{attribute 'enable_dynamic_creation'}
FUNCTION_BLOCK FB_DBTransactionHandler
VAR_INPUT
	ProjectDBDefs : IProjectDBDefs; //Instance of the custom database FB for this database
END_VAR
VAR_OUTPUT
END_VAR
VAR
	//Property backing variables
	_JRSQLNetId : T_AmsNetID;
	_JRSQLPort : T_AmsPort;
	_DBServer : POINTER TO fb_dbserver;
	_Busy : BOOL;
	_Done : BOOL;
	_Error : BOOL;
	_ErrorId : UINT;	
	_ErrorText : STRING;
	
	//'Framework'
	bFirstScan: BOOL := TRUE;
	tmrState:  TON;

	nState:	UDINT	:= 0;
	nNextState:	UDINT	:= 0;
	bFirstEntry: BOOL;	
	
	//Locals
	Triggered : BOOL := FALSE;
	DataReturn : BOOL := FALSE;
	
	spName :STRING;
	spData: pvoid;
	spDataSize:UDINT;
	
	spDefinition : DBSPDefinition;
	spCallResult : DBSPCallResult;
	
	TransmitBuffer : POINTER TO BYTE;
	TransmitSize : UINT;
	ReceiveBuffer : POINTER TO BYTE;
	ReceiveSize : UINT;
	
	LastProcessTime : TIME;
		
	fbADSReadWrite: ADSRDWRTEX;

END_VAR
VAR CONSTANT
	cJRSQLTimeout : TIME := T#10S;
	cJRSQLCommandExecute : UDINT := 16#1000;
END_VAR

IF bFirstScan THEN
	nNextState:=0;
	nState:=9999;
	
	fbADSReadWrite(NETID:=_JRSQLNetId,PORT:=_JRSQLPort,WRTRD:=FALSE,TMOUT:=cJRSQLTimeout);
	bFirstScan := FALSE;
END_IF

//state machine	
IF nState <> nNextState THEN
	bFirstEntry := TRUE;
	nState := nNextState;
ELSE
	bFirstEntry := FALSE;
END_IF

tmrState(IN:=(NOT bFirstEntry), PT:=T#20S);

CASE nState OF
0:
	IF bFirstEntry THEN
		_Error:=FALSE;
		_ErrorId := 16#0;
		_ErrorText := '';
		_Done:=FALSE;
	END_IF

	IF Triggered THEN
		IF _DBServer^.Connected THEN
			nNextState := 40;
		ELSE
			nNextState := 10;
		END_IF
	END_IF
	
10://wait for connection
	IF (_DBServer^.Connected) THEN
		nNextState := 0;
	ELSIF tmrState.ET > cJRSQLTimeout THEN
		_ErrorText:='JRSQL connection timeout';		
		_ErrorId := 16#1;
		_Error:=TRUE;
		nNextState	:= 999;
 	END_IF

//States combined to get rid of scan delays	
40: //Call JRSQL
	IF bFirstEntry THEN
		IF(ProjectDBDefs.GetSPDef(spName, ADR(spDefinition))) THEN
			TransmitSize := SIZEOF(DBSPDefinition) + spDefinition.InputParamSize;
			ReceiveSize := SIZEOF(DBSPCallResult) + spDefinition.OutputParamSize;

			IF (spDataSize = spDefinition.InputParamSize+spDefinition.OutputParamSize) THEN
				;
			ELSE
				_ErrorText := CONCAT('Procedure data size mismatch. Expected: ',CONCAT(UINT_TO_STRING(spDefinition.InputParamSize+spDefinition.OutputParamSize),CONCAT(' Got: ',UDINT_TO_STRING(spDataSize))));
				_ErrorId:= 16#3;
				_Error:=TRUE;
				nNextState := 999;
			END_IF
		ELSE 
			_ErrorText:='Stored procedure not found';		
			_ErrorId := 16#2;
			_Error:=TRUE;
			nNextState	:= 999;		
		END_IF	
	
		IF (NOT _Error) THEN
			//Allocate buffers
			TransmitSize := SIZEOF(DBSPDefinition) + spDefinition.InputParamSize;
			TransmitBuffer := __NEW(BYTE, TransmitSize);
			MEMSET(TransmitBuffer,0,TransmitSize);
			ReceiveSize := SIZEOF(DBSPCallResult) + spDefinition.OutputParamSize;
			ReceiveBuffer := __NEW(BYTE, ReceiveSize);
			MEMSET(ReceiveBuffer,0,ReceiveSize);
		
			memcpy(TransmitBuffer,ADR(spDefinition),SIZEOF(DBSPDefinition));
			memcpy((TransmitBuffer + SIZEOF(DBSPDefinition)),spData,spDefinition.InputParamSize);
		END_IF
	END_IF

	IF (NOT _Error) THEN
		
		fbADSReadWrite(WRTRD:=TRUE, IDXGRP:=cJRSQLCommandExecute, WRITELEN:=TransmitSize, SRCADDR:= TransmitBuffer, READLEN:=ReceiveSize, DESTADDR:= ReceiveBuffer);

		IF NOT fbADSReadWrite.Busy THEN
			IF NOT fbADSReadWrite.ERR THEN
				memcpy(ADR(spCallResult),ReceiveBuffer,SIZEOF(DBSPCallResult));
			
				IF spCallResult.Result <> 1 THEN
					//Error returned by JRSQL
					_ErrorText := CONCAT('JRSQL error: ',spCallResult.ResultString);
					_ErrorId:= 16#1000 + spCallResult.Result;
					_Error:=TRUE;
					nNextState := 999;
				ELSE
					//Copy result to caller
					memcpy(spData+spDefinition.InputParamSize,ReceiveBuffer+SIZEOF(DBSPCallResult),spDefinition.OutputParamSize);
					LastProcessTime := spCallResult.ProcessTime;
					_Done:=TRUE;
					nNextState := 999;		
				END_IF
			ELSE
				IF fbADSReadWrite.ERRID = 1861 THEN
					_ErrorText := 'JRSQL response timeout';
					_ErrorId:= 16#8;
					_Error:=TRUE;
					nNextState := 999;	
				ELSE
					_ErrorText := Concat('Error communicating to JRSQL: ', UDINT_TO_STRING(fbADSReadWrite.ERRID));
					_ErrorId:= 16#9;
					_Error:=TRUE;
					nNextState := 999;	
				END_IF
			END_IF
		END_IF
	
		IF (nState <> nNextState) THEN
			fbADSReadWrite(WRTRD:=FALSE);
			__DELETE(TransmitBuffer);
			__DELETE(ReceiveBuffer);
		END_IF
	
	END_IF
	
999:
	IF bFirstEntry THEN
		IF NOT _Error THEN
			_Done:=TRUE;
		END_IF
	END_IF
	
	IF NOT Triggered THEN
		nNextState	:= 0;	
	END_IF

END_CASE	

_Busy := (nState <> 0);
Triggered:=FALSE;
DataReturn:=FALSE;

PROPERTY Busy : bool
GET
Busy := _Busy;
END_GET
END_PROPERTY

PROPERTY Done : bool
GET
Done := _Done;
END_GET
END_PROPERTY

PROPERTY Error : bool
GET
Error := _Error;
END_GET
END_PROPERTY

PROPERTY ErrorId : UDINT
GET
ErrorId := _ErrorId;
END_GET
END_PROPERTY

PROPERTY ErrorText : STRING
GET
ErrorText := _ErrorText;
END_GET
END_PROPERTY

METHOD ExecuteSP : BOOL
VAR_INPUT
	bForeground : BOOL;
	sSPName : STRING;
	pData : pvoid;
	nDataSize : UDINT;
END_VAR
VAR
	BackgroundItem : POINTER TO DBBackgroundItem;
	
	
END_VAR
IF bForeground THEN
	//execute in process
	IF NOT busy THEN
		//first time call, set data
		spName := sSPName;
		spData := pData;
		spDataSize := nDataSize;
	ELSE
		//subsequent call
	
	END_IF

	Triggered:=TRUE;
	DataReturn:=FALSE;
	ExecuteSP:=(_Done OR _Error);
ELSE
	//build a new item to disassociate from the caller
	BackgroundItem:= __NEW(DBBackgroundItem);
	BackgroundItem^.SPName := sSPName;
	BackgroundItem^.DataSize := nDataSize;
	memcpy(ADR(BackgroundItem^.Data),pData,nDataSize);
	
	//Pass it off to the background fifo	
	IF NOT (_DBServer^.AddBackgroundItem(BackgroundItem)) THEN
		//add failed, clear the memory

		__DELETE(BackgroundItem);
	END_IF
	
	ExecuteSP:=TRUE;
END_IF
END_METHOD

METHOD FB_init : BOOL
VAR_INPUT
	bInitRetains : BOOL; // if TRUE, the retain variables are initialized (warm start / cold start)
	bInCopyCode : BOOL;  // if TRUE, the instance afterwards gets moved into the copy code (online change)
	
	pDBServer : POINTER TO FB_DBServer; //Instance of the custom database FB for this database
	JRSQLNetId : T_AmsNetID := ''; //AMS address of JRSQL
	JRSQLPort : T_AmsPort := 2020; //AMS port of JRSQL
	ProjectDBDefs : IProjectDBDefs; //Project database config
	
END_VAR
_DBServer := pDBServer;
_JRSQLNetId := JRSQLNetId;
_JRSQLPort := JRSQLPort;
THIS^.ProjectDBDefs := ProjectDBDefs;

IF bInitRetains THEN
	bFirstScan := TRUE;
END_IF
END_METHOD

END_FUNCTION_BLOCK

(* stored: Version 1.1.0.1, ProductVersion 3.1.4024.6
   POU FB_DBTransactionHandler: Id {701ed8f0-97e9-43b4-b1db-6fc299a99a7b}, SpecialFunc None
   Property Busy: Id {f1ddb760-7bb3-4dcd-b84d-873d0192d8f5}
   Get Get: Id {626c016b-ecd5-4098-9bcb-b1a7335cd3a5}
   Property Done: Id {7b7a4b19-a4f9-47cf-bea9-02618afbc18d}
   Get Get: Id {e1f21e46-f346-4627-9b10-69b059d736da}
   Property Error: Id {fd745fdc-4fa3-451b-8cb3-e62b0590349d}
   Get Get: Id {f0e0774e-80cf-4dcc-83fa-99f6dfb518ae}
   Property ErrorId: Id {cb7cd9e7-60d0-4f1b-b380-1b1a7187bee3}
   Get Get: Id {79105363-ebeb-443d-8b4d-6ead43893a21}
   Property ErrorText: Id {6b8e88de-7b14-4647-ade8-fb4e9620db9c}
   Get Get: Id {cec451ed-c226-412b-8581-fd29f3f71216}
   Method ExecuteSP: Id {8b7c64c6-825c-456d-a298-9d21c2818ee5}
   Method FB_init: Id {eb2e57a6-0d93-4e26-8da9-9f4dead7454c} *)
